{attribute 'GeneratedUsingTerminal: EL6690-0002-0000'}
{attribute addProperty BoxType "EL6690-0002-0000"}
{attribute addProperty Id "StatusAT %I*Status_D30DC33F1InputsEMPTY_STRUCTURE0OutputsEMPTY_STRUCTURE0WcStateAT %I*WcState_9091E0EB2InfoDataAT %I*InfoData_6F19DB2B2"}
{attribute addProperty CRC "895781002"}
{attribute addProperty Size "5"}
TYPE EL6690_3564888A EXTENDS EtcSlaveTerminalBase_947E5A46 :
STRUCT
	{attribute addProperty Name "Status"}
	Status : Status_D30DC33F;
	{attribute addProperty Name "Inputs"}
	Inputs : EMPTY_STRUCTURE;
	{attribute addProperty Name "Outputs"}
	Outputs : EMPTY_STRUCTURE;
	{attribute addProperty Name "WcState"}
	WcState : WcState_9091E0EB;
	{attribute addProperty Name "InfoData"}
	InfoData : InfoData_6F19DB2B;
END_STRUCT
END_TYPE

(* stored: Version 1.2.0.0, ProductVersion 3.1.4024.9
   DUT EL6690_3564888A: Id {f73ac524-5dda-427e-b0f1-178661525daf} *)
